FUNCTION BFT_TO_MS : REAL
VAR_INPUT
	BFT : INT;
END_VAR


(*
version 1.0	12. jun 2008
programmer 	hugo
tested by		oscdat

this function converts wind speed from beaufort to m/s
*)


BFT_TO_MS := LREAL_TO_REAL(EXPT(BFT, 1.5) * 0.836);


(* revision history
hm	12. 6. 2008		rev 1.0
	original version

*)

END_FUNCTION

(* stored: Version 1.1.0.1
   POU BFT_TO_MS: Id {10811f22-67d5-46e7-8f92-2cf79e120d0e}, SpecialFunc None *)
